// TIA Portal V20 export
TYPE "typeDataToSafety"
// Information sent from the standard program to the safety program
// stored: Access Published, IsFailsafeCompliant true, Namespace Safety
   STRUCT
      ackSafetyFromHmi : Int;   // Acknowledge variable from operator control or monitoring system
      ackSafetyGlobal : Bool;   // Acknowledge command to ack all safety
      ackFromUnit1 : Bool;   // Acknowledge command coming from Unit 1
      ackSafetyFromMobileHMI : Bool;   // Acknowledge command coming from Mobile Panel
      resetSafetyFromMobileHMI : Bool;   // Reset command coming from Mobile Panel
      connectionBoxID_1 : Int;   // Mobile Panel Connection Box ID (extend list as needed)
      connectionBoxID_2 : Int;   // Mobile Panel Connection Box ID (extend list as needed)
      MobilePanelConnected : Bool;   // TRUE: connection box is connected
      MobilePannelPermissions : Bool;
      "PhmiNo1.Connected" : Bool;
      "PhmiNo2.Connected" : Bool;
      KeyBoxStatus : Int;
      DeselectBA30 : Bool;   // BA30 is not selected and no supply part
      DeselectBA40 : Bool;   // BA40 is not selected and no supply part
      DeselectBA15 : Bool;   // BA15 is not selected and no supply part
      DeselectBA60 : Bool;   // BA60 is not selected and no supply part
      PowerOnCommand : Bool;   // Power On Command
      leftUnwinderRadius : Int;
      rightUnwinderRadius : Int;
      PhmiCommunicationOK : Bool;   // PHMI Communication OK
      allBrakeTesting : "Safety.typeBrakeTest";
      Unwinder_Left_DiaData : "Safety.typeSafetyDia";
      Unwinder_Right_DiaData : "Safety.typeSafetyDia";
      FrameCoverSensor : "Safety.SensorStatus";
      unitMode : "Safety.typeUnitMode";   // Current mode of the unit
      unitState : "Safety.typeUnitStatus";   // Current States of the unit
      winderUsed : "Safety.typeWinderUseMode";
      GateCutter : "Safety.typeFdoorCommands";   // Gate Control Cutter
      GateMagazine : "Safety.typeFdoorCommands";   // Gate Control Magazine
      GateConveyor : "Safety.typeFdoorCommands";   // Gate Control Conveyor
      GateCentralAisle : "Safety.typeFdoorCommands";
      scrapBox1Interface : "Safety.typeScrapBoxMonitoring";
      OpLampStatus : "Safety.typeOpLampStatus";
      clock : "Safety.typeGlobalClockMem";
   END_STRUCT;
END_TYPE
